// TIA Portal V19 export
FUNCTION "SUB_OUTPUT" : Void   // FC9, LAD
{ S7_Optimized_Access := 'TRUE' }
// stored: SetENOAutomatically false
BEGIN

REGION Network 1: "MGF FEED PUMP WORKING"
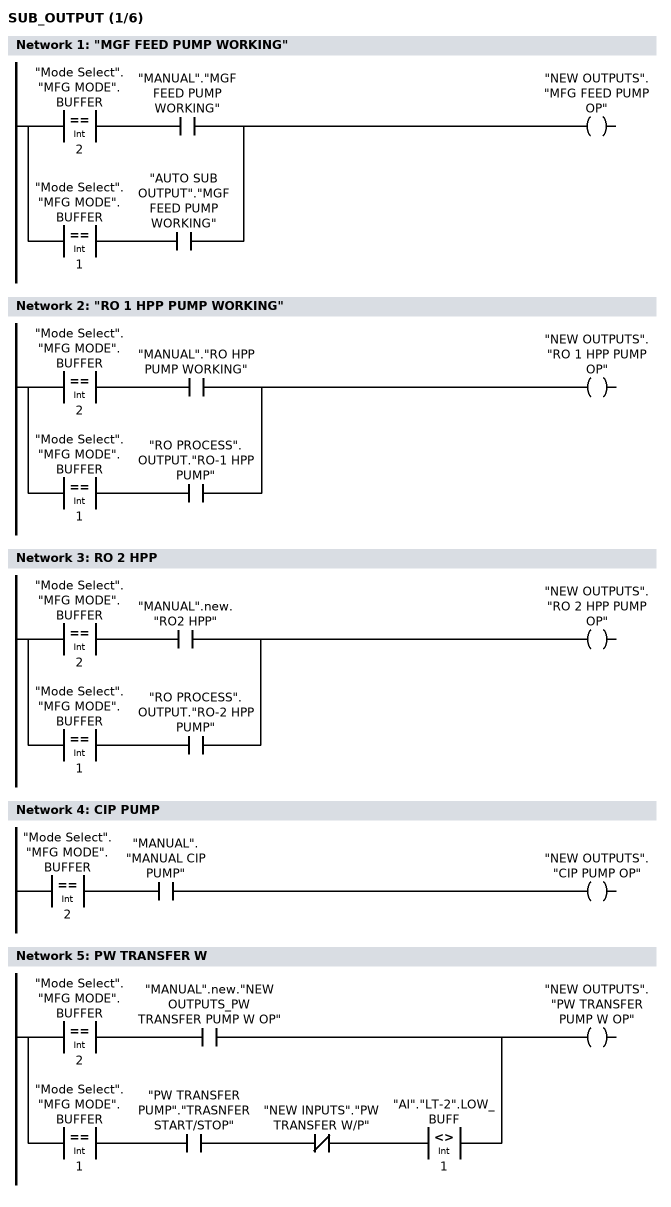
   RUNG wire#powerrail
      { S7_Templates := "SrcType := Int" } EQ_Contact(in1 := "Mode Select"."MFG MODE".BUFFER, in2 := 2)
      Contact( "MANUAL"."MGF FEED PUMP WORKING" )
      wire#w1
      Coil( "NEW OUTPUTS"."MFG FEED PUMP OP" )
   END_RUNG
   RUNG wire#powerrail
      { S7_Templates := "SrcType := Int" } EQ_Contact(in1 := "Mode Select"."MFG MODE".BUFFER, in2 := 1)
      Contact( "AUTO SUB OUTPUT"."MGF FEED PUMP WORKING" )
   END_RUNG wire#w1
   // the same network as SCL:
   "NEW OUTPUTS"."MFG FEED PUMP OP" := (("Mode Select"."MFG MODE".BUFFER = 2) AND "MANUAL"."MGF FEED PUMP WORKING") OR (("Mode Select"."MFG MODE".BUFFER = 1) AND "AUTO SUB OUTPUT"."MGF FEED PUMP WORKING");
END_REGION

REGION Network 2: "RO 1 HPP PUMP WORKING"
   RUNG wire#powerrail
      { S7_Templates := "SrcType := Int" } EQ_Contact(in1 := "Mode Select"."MFG MODE".BUFFER, in2 := 2)
      Contact( "MANUAL"."RO HPP PUMP WORKING" )
      wire#w1
      Coil( "NEW OUTPUTS"."RO 1 HPP PUMP OP" )
   END_RUNG
   RUNG wire#powerrail
      { S7_Templates := "SrcType := Int" } EQ_Contact(in1 := "Mode Select"."MFG MODE".BUFFER, in2 := 1)
      Contact( "RO PROCESS".OUTPUT."RO-1 HPP PUMP" )
   END_RUNG wire#w1
   // the same network as SCL:
   "NEW OUTPUTS"."RO 1 HPP PUMP OP" := (("Mode Select"."MFG MODE".BUFFER = 2) AND "MANUAL"."RO HPP PUMP WORKING") OR (("Mode Select"."MFG MODE".BUFFER = 1) AND "RO PROCESS".OUTPUT."RO-1 HPP PUMP");
END_REGION

REGION Network 3: RO 2 HPP
   RUNG wire#powerrail
      { S7_Templates := "SrcType := Int" } EQ_Contact(in1 := "Mode Select"."MFG MODE".BUFFER, in2 := 2)
      Contact( "MANUAL".new."RO2 HPP" )
      wire#w1
      Coil( "NEW OUTPUTS"."RO 2 HPP PUMP OP" )
   END_RUNG
   RUNG wire#powerrail
      { S7_Templates := "SrcType := Int" } EQ_Contact(in1 := "Mode Select"."MFG MODE".BUFFER, in2 := 1)
      Contact( "RO PROCESS".OUTPUT."RO-2 HPP PUMP" )
   END_RUNG wire#w1
   // the same network as SCL:
   "NEW OUTPUTS"."RO 2 HPP PUMP OP" := (("Mode Select"."MFG MODE".BUFFER = 2) AND "MANUAL".new."RO2 HPP") OR (("Mode Select"."MFG MODE".BUFFER = 1) AND "RO PROCESS".OUTPUT."RO-2 HPP PUMP");
END_REGION

REGION Network 4: CIP PUMP
   RUNG wire#powerrail
      { S7_Templates := "SrcType := Int" } EQ_Contact(in1 := "Mode Select"."MFG MODE".BUFFER, in2 := 2)
      Contact( "MANUAL"."MANUAL CIP PUMP" )
      Coil( "NEW OUTPUTS"."CIP PUMP OP" )
   END_RUNG
   // the same network as SCL:
   "NEW OUTPUTS"."CIP PUMP OP" := ("Mode Select"."MFG MODE".BUFFER = 2) AND "MANUAL"."MANUAL CIP PUMP";
END_REGION

REGION Network 5: PW TRANSFER W
   RUNG wire#powerrail
      { S7_Templates := "SrcType := Int" } EQ_Contact(in1 := "Mode Select"."MFG MODE".BUFFER, in2 := 2)
      Contact( "MANUAL".new."NEW OUTPUTS_PW TRANSFER PUMP W OP" )
      wire#w1
      Coil( "NEW OUTPUTS"."PW TRANSFER PUMP W OP" )
   END_RUNG
   RUNG wire#powerrail
      { S7_Templates := "SrcType := Int" } EQ_Contact(in1 := "Mode Select"."MFG MODE".BUFFER, in2 := 1)
      Contact( "PW TRANSFER PUMP"."TRASNFER START/STOP" )
      I_Contact( "NEW INPUTS"."PW TRANSFER W/P" )
      { S7_Templates := "SrcType := Int" } NE_Contact(in1 := "AI"."LT-2".LOW_BUFF, in2 := 1)
   END_RUNG wire#w1
   // the same network as SCL:
   "NEW OUTPUTS"."PW TRANSFER PUMP W OP" := (("Mode Select"."MFG MODE".BUFFER = 2) AND "MANUAL".new."NEW OUTPUTS_PW TRANSFER PUMP W OP") OR (("Mode Select"."MFG MODE".BUFFER = 1) AND "PW TRANSFER PUMP"."TRASNFER START/STOP" AND NOT "NEW INPUTS"."PW TRANSFER W/P" AND ("AI"."LT-2".LOW_BUFF <> 1));
END_REGION

REGION Network 6: PW TRANSFER S
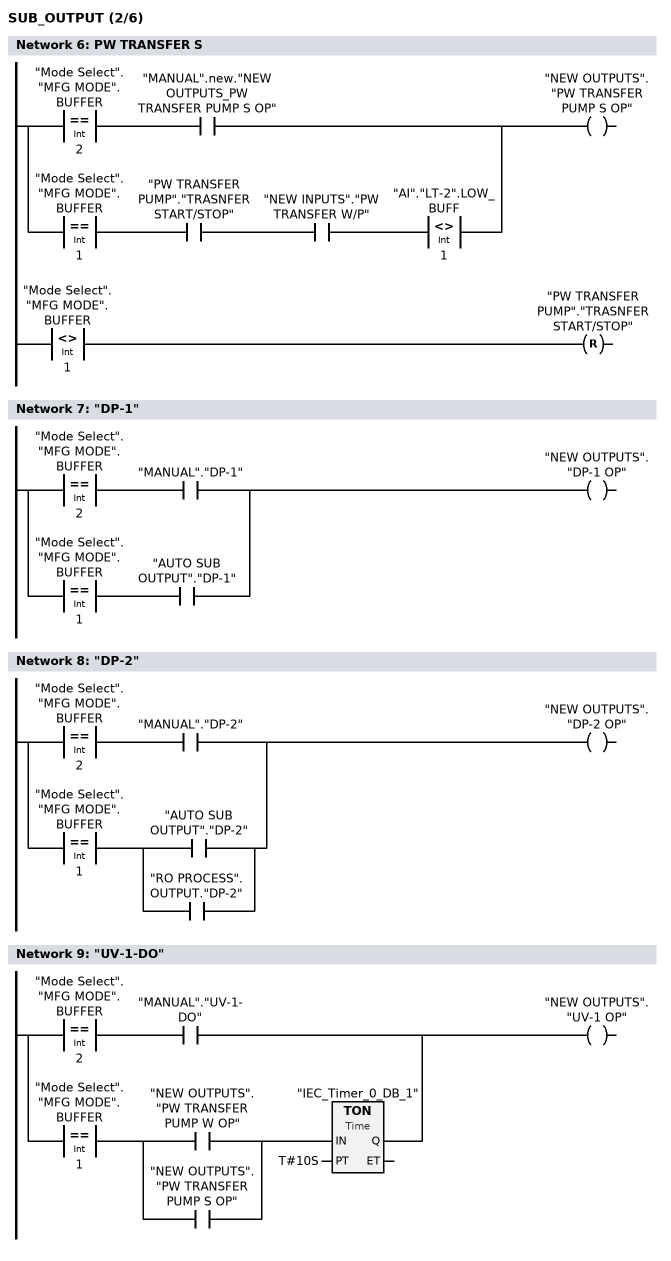
   RUNG wire#powerrail
      { S7_Templates := "SrcType := Int" } EQ_Contact(in1 := "Mode Select"."MFG MODE".BUFFER, in2 := 2)
      Contact( "MANUAL".new."NEW OUTPUTS_PW TRANSFER PUMP S OP" )
      wire#w1
      Coil( "NEW OUTPUTS"."PW TRANSFER PUMP S OP" )
   END_RUNG
   RUNG wire#powerrail
      { S7_Templates := "SrcType := Int" } EQ_Contact(in1 := "Mode Select"."MFG MODE".BUFFER, in2 := 1)
      Contact( "PW TRANSFER PUMP"."TRASNFER START/STOP" )
      Contact( "NEW INPUTS"."PW TRANSFER W/P" )
      { S7_Templates := "SrcType := Int" } NE_Contact(in1 := "AI"."LT-2".LOW_BUFF, in2 := 1)
   END_RUNG wire#w1
   RUNG wire#powerrail
      { S7_Templates := "SrcType := Int" } NE_Contact(in1 := "Mode Select"."MFG MODE".BUFFER, in2 := 1)
      R_Coil( "PW TRANSFER PUMP"."TRASNFER START/STOP" )
   END_RUNG
   // the same network as SCL:
   "NEW OUTPUTS"."PW TRANSFER PUMP S OP" := (("Mode Select"."MFG MODE".BUFFER = 2) AND "MANUAL".new."NEW OUTPUTS_PW TRANSFER PUMP S OP") OR (("Mode Select"."MFG MODE".BUFFER = 1) AND "PW TRANSFER PUMP"."TRASNFER START/STOP" AND "NEW INPUTS"."PW TRANSFER W/P" AND ("AI"."LT-2".LOW_BUFF <> 1));
   IF "Mode Select"."MFG MODE".BUFFER <> 1 THEN "PW TRANSFER PUMP"."TRASNFER START/STOP" := FALSE; END_IF;
END_REGION

REGION Network 7: "DP-1"
   RUNG wire#powerrail
      { S7_Templates := "SrcType := Int" } EQ_Contact(in1 := "Mode Select"."MFG MODE".BUFFER, in2 := 2)
      Contact( "MANUAL"."DP-1" )
      wire#w1
      Coil( "NEW OUTPUTS"."DP-1 OP" )
   END_RUNG
   RUNG wire#powerrail
      { S7_Templates := "SrcType := Int" } EQ_Contact(in1 := "Mode Select"."MFG MODE".BUFFER, in2 := 1)
      Contact( "AUTO SUB OUTPUT"."DP-1" )
   END_RUNG wire#w1
   // the same network as SCL:
   "NEW OUTPUTS"."DP-1 OP" := (("Mode Select"."MFG MODE".BUFFER = 2) AND "MANUAL"."DP-1") OR (("Mode Select"."MFG MODE".BUFFER = 1) AND "AUTO SUB OUTPUT"."DP-1");
END_REGION

REGION Network 8: "DP-2"
   RUNG wire#powerrail
      { S7_Templates := "SrcType := Int" } EQ_Contact(in1 := "Mode Select"."MFG MODE".BUFFER, in2 := 2)
      Contact( "MANUAL"."DP-2" )
      wire#w1
      Coil( "NEW OUTPUTS"."DP-2 OP" )
   END_RUNG
   RUNG wire#powerrail
      { S7_Templates := "SrcType := Int" } EQ_Contact(in1 := "Mode Select"."MFG MODE".BUFFER, in2 := 1)
      wire#w2
      Contact( "AUTO SUB OUTPUT"."DP-2" )
   END_RUNG wire#w1
   RUNG wire#w2
      Contact( "RO PROCESS".OUTPUT."DP-2" )
   END_RUNG wire#w1
   // the same network as SCL:
   "NEW OUTPUTS"."DP-2 OP" := (("Mode Select"."MFG MODE".BUFFER = 2) AND "MANUAL"."DP-2") OR (("Mode Select"."MFG MODE".BUFFER = 1) AND ("AUTO SUB OUTPUT"."DP-2" OR "RO PROCESS".OUTPUT."DP-2"));
END_REGION

REGION Network 9: "UV-1-DO"
   RUNG wire#powerrail
      { S7_Templates := "SrcType := Int" } EQ_Contact(in1 := "Mode Select"."MFG MODE".BUFFER, in2 := 2)
      Contact( "MANUAL"."UV-1-DO" )
      wire#w1
      Coil( "NEW OUTPUTS"."UV-1 OP" )
   END_RUNG
   RUNG wire#powerrail
      { S7_Templates := "SrcType := Int" } EQ_Contact(in1 := "Mode Select"."MFG MODE".BUFFER, in2 := 1)
      wire#w2
      Contact( "NEW OUTPUTS"."PW TRANSFER PUMP W OP" )
      wire#w3
      { S7_Templates := "time_type := Time" } "IEC_Timer_0_DB_1".TON(pt := T#10S, et =>)
   END_RUNG wire#w1
   RUNG wire#w2
      Contact( "NEW OUTPUTS"."PW TRANSFER PUMP S OP" )
   END_RUNG wire#w3
   // the same network as SCL:
   "IEC_Timer_0_DB_1".TON(IN := ("Mode Select"."MFG MODE".BUFFER = 1) AND ("NEW OUTPUTS"."PW TRANSFER PUMP W OP" OR "NEW OUTPUTS"."PW TRANSFER PUMP S OP"),
                          PT := T#10S);
   "NEW OUTPUTS"."UV-1 OP" := (("Mode Select"."MFG MODE".BUFFER = 2) AND "MANUAL"."UV-1-DO") OR "IEC_Timer_0_DB_1".Q;
END_REGION

REGION Network 10: "PSFV-1 – OPEN"
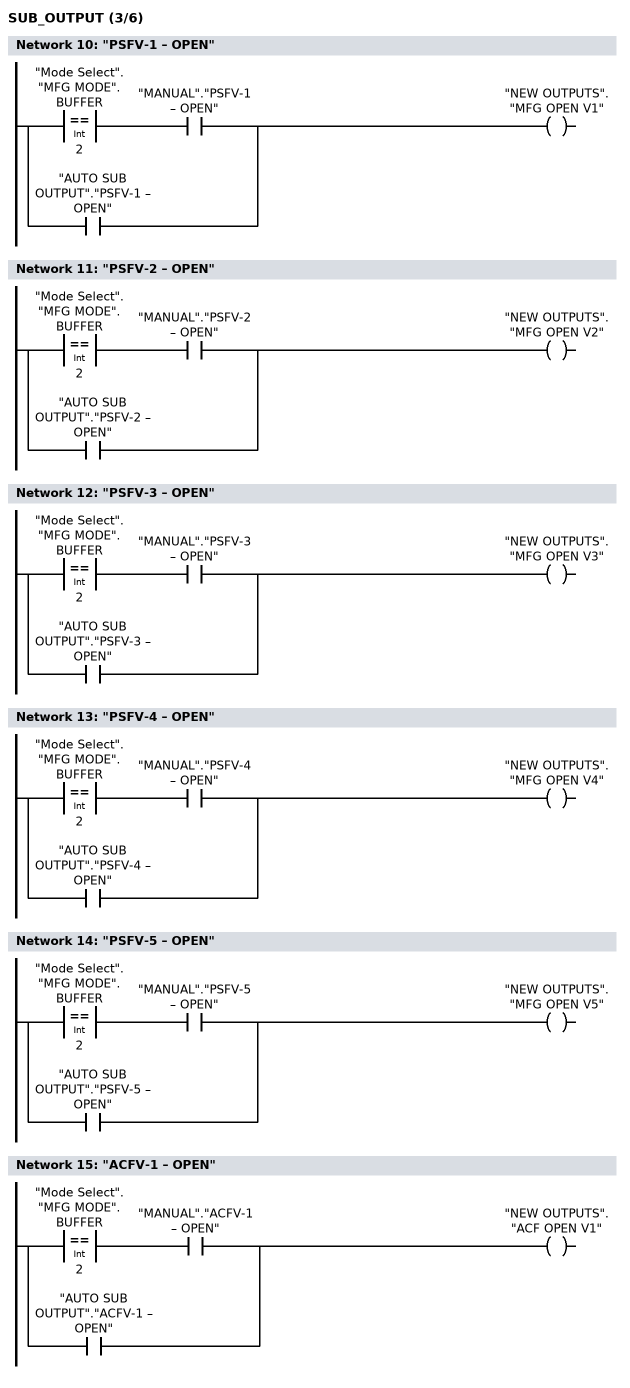
   RUNG wire#powerrail
      { S7_Templates := "SrcType := Int" } EQ_Contact(in1 := "Mode Select"."MFG MODE".BUFFER, in2 := 2)
      Contact( "MANUAL"."PSFV-1 – OPEN" )
      wire#w1
      Coil( "NEW OUTPUTS"."MFG OPEN V1" )
   END_RUNG
   RUNG wire#powerrail
      Contact( "AUTO SUB OUTPUT"."PSFV-1 – OPEN" )
   END_RUNG wire#w1
   // the same network as SCL:
   "NEW OUTPUTS"."MFG OPEN V1" := (("Mode Select"."MFG MODE".BUFFER = 2) AND "MANUAL"."PSFV-1 – OPEN") OR "AUTO SUB OUTPUT"."PSFV-1 – OPEN";
END_REGION

REGION Network 11: "PSFV-2 – OPEN"
   RUNG wire#powerrail
      { S7_Templates := "SrcType := Int" } EQ_Contact(in1 := "Mode Select"."MFG MODE".BUFFER, in2 := 2)
      Contact( "MANUAL"."PSFV-2 – OPEN" )
      wire#w1
      Coil( "NEW OUTPUTS"."MFG OPEN V2" )
   END_RUNG
   RUNG wire#powerrail
      Contact( "AUTO SUB OUTPUT"."PSFV-2 – OPEN" )
   END_RUNG wire#w1
   // the same network as SCL:
   "NEW OUTPUTS"."MFG OPEN V2" := (("Mode Select"."MFG MODE".BUFFER = 2) AND "MANUAL"."PSFV-2 – OPEN") OR "AUTO SUB OUTPUT"."PSFV-2 – OPEN";
END_REGION

REGION Network 12: "PSFV-3 – OPEN"
   RUNG wire#powerrail
      { S7_Templates := "SrcType := Int" } EQ_Contact(in1 := "Mode Select"."MFG MODE".BUFFER, in2 := 2)
      Contact( "MANUAL"."PSFV-3 – OPEN" )
      wire#w1
      Coil( "NEW OUTPUTS"."MFG OPEN V3" )
   END_RUNG
   RUNG wire#powerrail
      Contact( "AUTO SUB OUTPUT"."PSFV-3 – OPEN" )
   END_RUNG wire#w1
   // the same network as SCL:
   "NEW OUTPUTS"."MFG OPEN V3" := (("Mode Select"."MFG MODE".BUFFER = 2) AND "MANUAL"."PSFV-3 – OPEN") OR "AUTO SUB OUTPUT"."PSFV-3 – OPEN";
END_REGION

REGION Network 13: "PSFV-4 – OPEN"
   RUNG wire#powerrail
      { S7_Templates := "SrcType := Int" } EQ_Contact(in1 := "Mode Select"."MFG MODE".BUFFER, in2 := 2)
      Contact( "MANUAL"."PSFV-4 – OPEN" )
      wire#w1
      Coil( "NEW OUTPUTS"."MFG OPEN V4" )
   END_RUNG
   RUNG wire#powerrail
      Contact( "AUTO SUB OUTPUT"."PSFV-4 – OPEN" )
   END_RUNG wire#w1
   // the same network as SCL:
   "NEW OUTPUTS"."MFG OPEN V4" := (("Mode Select"."MFG MODE".BUFFER = 2) AND "MANUAL"."PSFV-4 – OPEN") OR "AUTO SUB OUTPUT"."PSFV-4 – OPEN";
END_REGION

REGION Network 14: "PSFV-5 – OPEN"
   RUNG wire#powerrail
      { S7_Templates := "SrcType := Int" } EQ_Contact(in1 := "Mode Select"."MFG MODE".BUFFER, in2 := 2)
      Contact( "MANUAL"."PSFV-5 – OPEN" )
      wire#w1
      Coil( "NEW OUTPUTS"."MFG OPEN V5" )
   END_RUNG
   RUNG wire#powerrail
      Contact( "AUTO SUB OUTPUT"."PSFV-5 – OPEN" )
   END_RUNG wire#w1
   // the same network as SCL:
   "NEW OUTPUTS"."MFG OPEN V5" := (("Mode Select"."MFG MODE".BUFFER = 2) AND "MANUAL"."PSFV-5 – OPEN") OR "AUTO SUB OUTPUT"."PSFV-5 – OPEN";
END_REGION

REGION Network 15: "ACFV-1 – OPEN"
   RUNG wire#powerrail
      { S7_Templates := "SrcType := Int" } EQ_Contact(in1 := "Mode Select"."MFG MODE".BUFFER, in2 := 2)
      Contact( "MANUAL"."ACFV-1 – OPEN" )
      wire#w1
      Coil( "NEW OUTPUTS"."ACF OPEN V1" )
   END_RUNG
   RUNG wire#powerrail
      Contact( "AUTO SUB OUTPUT"."ACFV-1 – OPEN" )
   END_RUNG wire#w1
   // the same network as SCL:
   "NEW OUTPUTS"."ACF OPEN V1" := (("Mode Select"."MFG MODE".BUFFER = 2) AND "MANUAL"."ACFV-1 – OPEN") OR "AUTO SUB OUTPUT"."ACFV-1 – OPEN";
END_REGION

REGION Network 16: "ACFV-2 – OPEN"
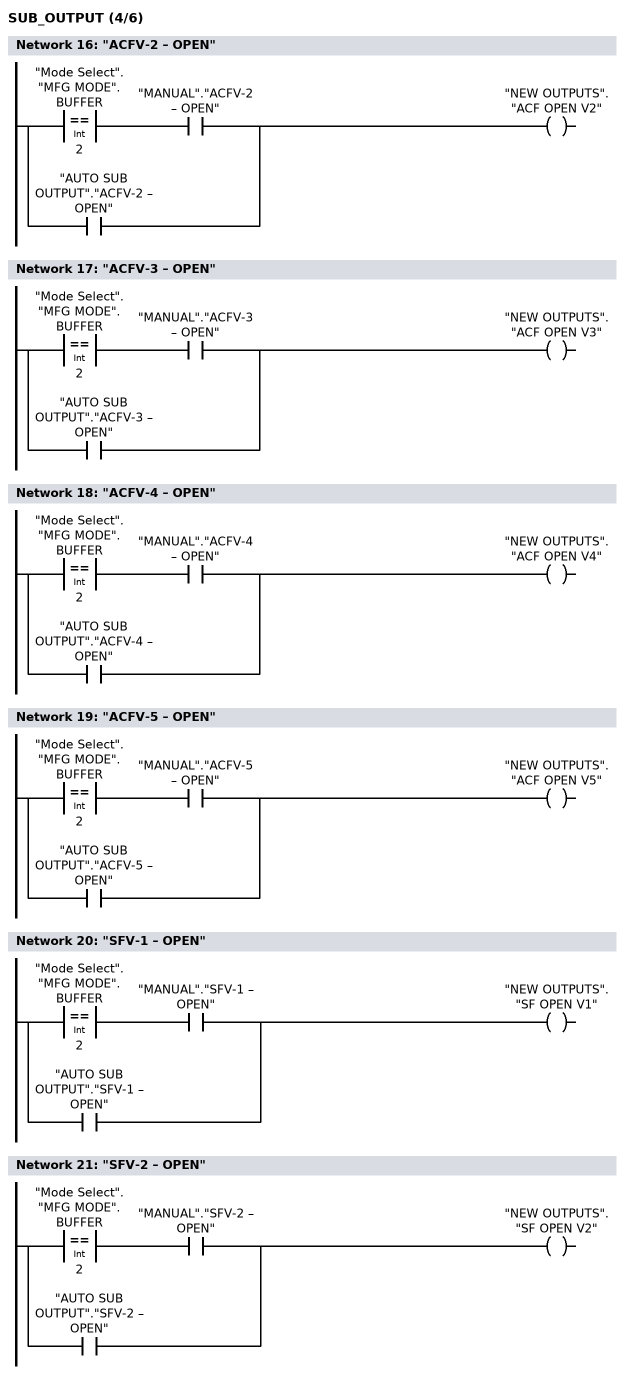
   RUNG wire#powerrail
      { S7_Templates := "SrcType := Int" } EQ_Contact(in1 := "Mode Select"."MFG MODE".BUFFER, in2 := 2)
      Contact( "MANUAL"."ACFV-2 – OPEN" )
      wire#w1
      Coil( "NEW OUTPUTS"."ACF OPEN V2" )
   END_RUNG
   RUNG wire#powerrail
      Contact( "AUTO SUB OUTPUT"."ACFV-2 – OPEN" )
   END_RUNG wire#w1
   // the same network as SCL:
   "NEW OUTPUTS"."ACF OPEN V2" := (("Mode Select"."MFG MODE".BUFFER = 2) AND "MANUAL"."ACFV-2 – OPEN") OR "AUTO SUB OUTPUT"."ACFV-2 – OPEN";
END_REGION

REGION Network 17: "ACFV-3 – OPEN"
   RUNG wire#powerrail
      { S7_Templates := "SrcType := Int" } EQ_Contact(in1 := "Mode Select"."MFG MODE".BUFFER, in2 := 2)
      Contact( "MANUAL"."ACFV-3 – OPEN" )
      wire#w1
      Coil( "NEW OUTPUTS"."ACF OPEN V3" )
   END_RUNG
   RUNG wire#powerrail
      Contact( "AUTO SUB OUTPUT"."ACFV-3 – OPEN" )
   END_RUNG wire#w1
   // the same network as SCL:
   "NEW OUTPUTS"."ACF OPEN V3" := (("Mode Select"."MFG MODE".BUFFER = 2) AND "MANUAL"."ACFV-3 – OPEN") OR "AUTO SUB OUTPUT"."ACFV-3 – OPEN";
END_REGION

REGION Network 18: "ACFV-4 – OPEN"
   RUNG wire#powerrail
      { S7_Templates := "SrcType := Int" } EQ_Contact(in1 := "Mode Select"."MFG MODE".BUFFER, in2 := 2)
      Contact( "MANUAL"."ACFV-4 – OPEN" )
      wire#w1
      Coil( "NEW OUTPUTS"."ACF OPEN V4" )
   END_RUNG
   RUNG wire#powerrail
      Contact( "AUTO SUB OUTPUT"."ACFV-4 – OPEN" )
   END_RUNG wire#w1
   // the same network as SCL:
   "NEW OUTPUTS"."ACF OPEN V4" := (("Mode Select"."MFG MODE".BUFFER = 2) AND "MANUAL"."ACFV-4 – OPEN") OR "AUTO SUB OUTPUT"."ACFV-4 – OPEN";
END_REGION

REGION Network 19: "ACFV-5 – OPEN"
   RUNG wire#powerrail
      { S7_Templates := "SrcType := Int" } EQ_Contact(in1 := "Mode Select"."MFG MODE".BUFFER, in2 := 2)
      Contact( "MANUAL"."ACFV-5 – OPEN" )
      wire#w1
      Coil( "NEW OUTPUTS"."ACF OPEN V5" )
   END_RUNG
   RUNG wire#powerrail
      Contact( "AUTO SUB OUTPUT"."ACFV-5 – OPEN" )
   END_RUNG wire#w1
   // the same network as SCL:
   "NEW OUTPUTS"."ACF OPEN V5" := (("Mode Select"."MFG MODE".BUFFER = 2) AND "MANUAL"."ACFV-5 – OPEN") OR "AUTO SUB OUTPUT"."ACFV-5 – OPEN";
END_REGION

REGION Network 20: "SFV-1 – OPEN"
   RUNG wire#powerrail
      { S7_Templates := "SrcType := Int" } EQ_Contact(in1 := "Mode Select"."MFG MODE".BUFFER, in2 := 2)
      Contact( "MANUAL"."SFV-1 – OPEN" )
      wire#w1
      Coil( "NEW OUTPUTS"."SF OPEN V1" )
   END_RUNG
   RUNG wire#powerrail
      Contact( "AUTO SUB OUTPUT"."SFV-1 – OPEN" )
   END_RUNG wire#w1
   // the same network as SCL:
   "NEW OUTPUTS"."SF OPEN V1" := (("Mode Select"."MFG MODE".BUFFER = 2) AND "MANUAL"."SFV-1 – OPEN") OR "AUTO SUB OUTPUT"."SFV-1 – OPEN";
END_REGION

REGION Network 21: "SFV-2 – OPEN"
   RUNG wire#powerrail
      { S7_Templates := "SrcType := Int" } EQ_Contact(in1 := "Mode Select"."MFG MODE".BUFFER, in2 := 2)
      Contact( "MANUAL"."SFV-2 – OPEN" )
      wire#w1
      Coil( "NEW OUTPUTS"."SF OPEN V2" )
   END_RUNG
   RUNG wire#powerrail
      Contact( "AUTO SUB OUTPUT"."SFV-2 – OPEN" )
   END_RUNG wire#w1
   // the same network as SCL:
   "NEW OUTPUTS"."SF OPEN V2" := (("Mode Select"."MFG MODE".BUFFER = 2) AND "MANUAL"."SFV-2 – OPEN") OR "AUTO SUB OUTPUT"."SFV-2 – OPEN";
END_REGION

REGION Network 22: "SFV-3 – OPEN"
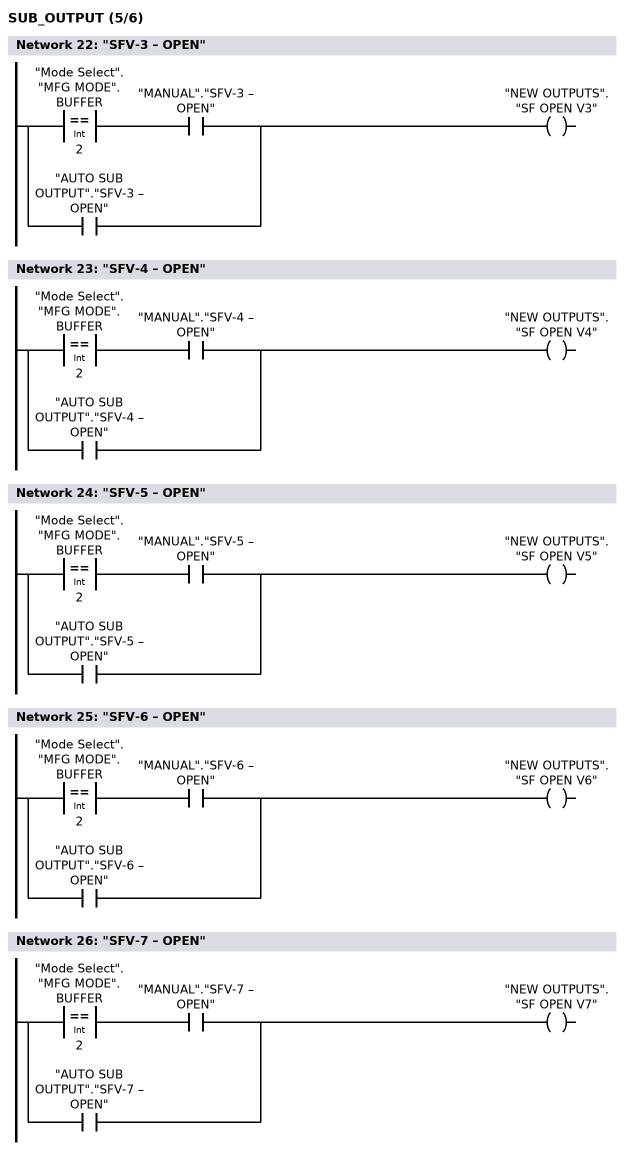
   RUNG wire#powerrail
      { S7_Templates := "SrcType := Int" } EQ_Contact(in1 := "Mode Select"."MFG MODE".BUFFER, in2 := 2)
      Contact( "MANUAL"."SFV-3 – OPEN" )
      wire#w1
      Coil( "NEW OUTPUTS"."SF OPEN V3" )
   END_RUNG
   RUNG wire#powerrail
      Contact( "AUTO SUB OUTPUT"."SFV-3 – OPEN" )
   END_RUNG wire#w1
   // the same network as SCL:
   "NEW OUTPUTS"."SF OPEN V3" := (("Mode Select"."MFG MODE".BUFFER = 2) AND "MANUAL"."SFV-3 – OPEN") OR "AUTO SUB OUTPUT"."SFV-3 – OPEN";
END_REGION

REGION Network 23: "SFV-4 – OPEN"
   RUNG wire#powerrail
      { S7_Templates := "SrcType := Int" } EQ_Contact(in1 := "Mode Select"."MFG MODE".BUFFER, in2 := 2)
      Contact( "MANUAL"."SFV-4 – OPEN" )
      wire#w1
      Coil( "NEW OUTPUTS"."SF OPEN V4" )
   END_RUNG
   RUNG wire#powerrail
      Contact( "AUTO SUB OUTPUT"."SFV-4 – OPEN" )
   END_RUNG wire#w1
   // the same network as SCL:
   "NEW OUTPUTS"."SF OPEN V4" := (("Mode Select"."MFG MODE".BUFFER = 2) AND "MANUAL"."SFV-4 – OPEN") OR "AUTO SUB OUTPUT"."SFV-4 – OPEN";
END_REGION

REGION Network 24: "SFV-5 – OPEN"
   RUNG wire#powerrail
      { S7_Templates := "SrcType := Int" } EQ_Contact(in1 := "Mode Select"."MFG MODE".BUFFER, in2 := 2)
      Contact( "MANUAL"."SFV-5 – OPEN" )
      wire#w1
      Coil( "NEW OUTPUTS"."SF OPEN V5" )
   END_RUNG
   RUNG wire#powerrail
      Contact( "AUTO SUB OUTPUT"."SFV-5 – OPEN" )
   END_RUNG wire#w1
   // the same network as SCL:
   "NEW OUTPUTS"."SF OPEN V5" := (("Mode Select"."MFG MODE".BUFFER = 2) AND "MANUAL"."SFV-5 – OPEN") OR "AUTO SUB OUTPUT"."SFV-5 – OPEN";
END_REGION

REGION Network 25: "SFV-6 – OPEN"
   RUNG wire#powerrail
      { S7_Templates := "SrcType := Int" } EQ_Contact(in1 := "Mode Select"."MFG MODE".BUFFER, in2 := 2)
      Contact( "MANUAL"."SFV-6 – OPEN" )
      wire#w1
      Coil( "NEW OUTPUTS"."SF OPEN V6" )
   END_RUNG
   RUNG wire#powerrail
      Contact( "AUTO SUB OUTPUT"."SFV-6 – OPEN" )
   END_RUNG wire#w1
   // the same network as SCL:
   "NEW OUTPUTS"."SF OPEN V6" := (("Mode Select"."MFG MODE".BUFFER = 2) AND "MANUAL"."SFV-6 – OPEN") OR "AUTO SUB OUTPUT"."SFV-6 – OPEN";
END_REGION

REGION Network 26: "SFV-7 – OPEN"
   RUNG wire#powerrail
      { S7_Templates := "SrcType := Int" } EQ_Contact(in1 := "Mode Select"."MFG MODE".BUFFER, in2 := 2)
      Contact( "MANUAL"."SFV-7 – OPEN" )
      wire#w1
      Coil( "NEW OUTPUTS"."SF OPEN V7" )
   END_RUNG
   RUNG wire#powerrail
      Contact( "AUTO SUB OUTPUT"."SFV-7 – OPEN" )
   END_RUNG wire#w1
   // the same network as SCL:
   "NEW OUTPUTS"."SF OPEN V7" := (("Mode Select"."MFG MODE".BUFFER = 2) AND "MANUAL"."SFV-7 – OPEN") OR "AUTO SUB OUTPUT"."SFV-7 – OPEN";
END_REGION

REGION Network 27: "AV-1 – OPEN"
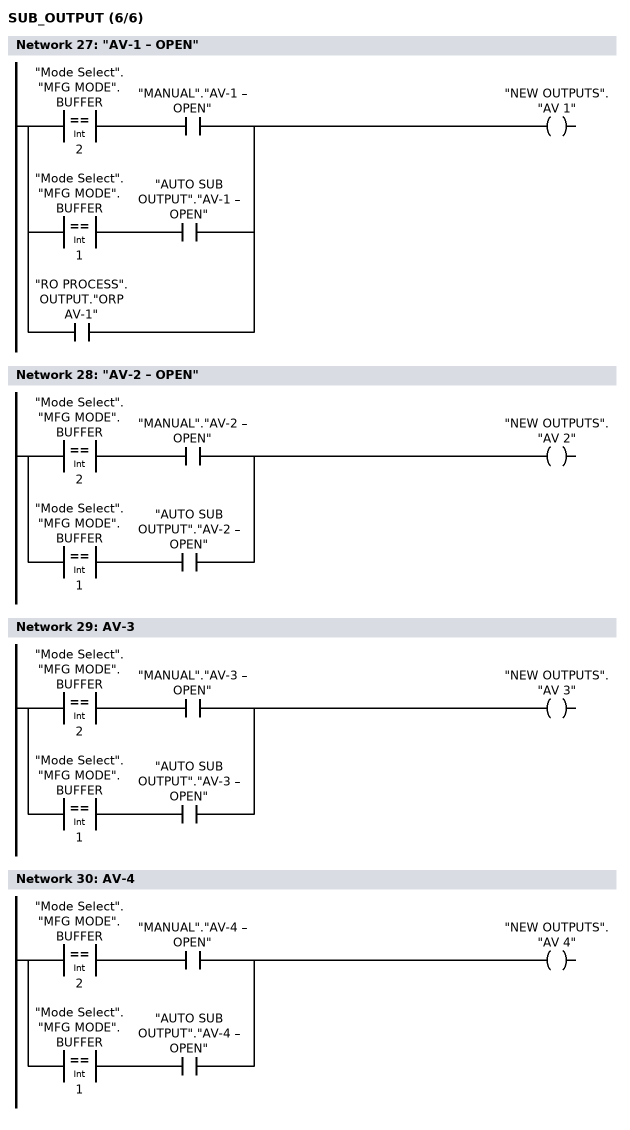
   RUNG wire#powerrail
      { S7_Templates := "SrcType := Int" } EQ_Contact(in1 := "Mode Select"."MFG MODE".BUFFER, in2 := 2)
      Contact( "MANUAL"."AV-1 – OPEN" )
      wire#w1
      Coil( "NEW OUTPUTS"."AV 1" )
   END_RUNG
   RUNG wire#powerrail
      { S7_Templates := "SrcType := Int" } EQ_Contact(in1 := "Mode Select"."MFG MODE".BUFFER, in2 := 1)
      Contact( "AUTO SUB OUTPUT"."AV-1 – OPEN" )
   END_RUNG wire#w1
   RUNG wire#powerrail
      Contact( "RO PROCESS".OUTPUT."ORP AV-1" )
   END_RUNG wire#w1
   // the same network as SCL:
   "NEW OUTPUTS"."AV 1" := (("Mode Select"."MFG MODE".BUFFER = 2) AND "MANUAL"."AV-1 – OPEN") OR (("Mode Select"."MFG MODE".BUFFER = 1) AND "AUTO SUB OUTPUT"."AV-1 – OPEN") OR "RO PROCESS".OUTPUT."ORP AV-1";
END_REGION

REGION Network 28: "AV-2 – OPEN"
   RUNG wire#powerrail
      { S7_Templates := "SrcType := Int" } EQ_Contact(in1 := "Mode Select"."MFG MODE".BUFFER, in2 := 2)
      Contact( "MANUAL"."AV-2 – OPEN" )
      wire#w1
      Coil( "NEW OUTPUTS"."AV 2" )
   END_RUNG
   RUNG wire#powerrail
      { S7_Templates := "SrcType := Int" } EQ_Contact(in1 := "Mode Select"."MFG MODE".BUFFER, in2 := 1)
      Contact( "AUTO SUB OUTPUT"."AV-2 – OPEN" )
   END_RUNG wire#w1
   // the same network as SCL:
   "NEW OUTPUTS"."AV 2" := (("Mode Select"."MFG MODE".BUFFER = 2) AND "MANUAL"."AV-2 – OPEN") OR (("Mode Select"."MFG MODE".BUFFER = 1) AND "AUTO SUB OUTPUT"."AV-2 – OPEN");
END_REGION

REGION Network 29: AV-3
   RUNG wire#powerrail
      { S7_Templates := "SrcType := Int" } EQ_Contact(in1 := "Mode Select"."MFG MODE".BUFFER, in2 := 2)
      Contact( "MANUAL"."AV-3 – OPEN" )
      wire#w1
      Coil( "NEW OUTPUTS"."AV 3" )
   END_RUNG
   RUNG wire#powerrail
      { S7_Templates := "SrcType := Int" } EQ_Contact(in1 := "Mode Select"."MFG MODE".BUFFER, in2 := 1)
      Contact( "AUTO SUB OUTPUT"."AV-3 – OPEN" )
   END_RUNG wire#w1
   // the same network as SCL:
   "NEW OUTPUTS"."AV 3" := (("Mode Select"."MFG MODE".BUFFER = 2) AND "MANUAL"."AV-3 – OPEN") OR (("Mode Select"."MFG MODE".BUFFER = 1) AND "AUTO SUB OUTPUT"."AV-3 – OPEN");
END_REGION

REGION Network 30: AV-4
   RUNG wire#powerrail
      { S7_Templates := "SrcType := Int" } EQ_Contact(in1 := "Mode Select"."MFG MODE".BUFFER, in2 := 2)
      Contact( "MANUAL"."AV-4 – OPEN" )
      wire#w1
      Coil( "NEW OUTPUTS"."AV 4" )
   END_RUNG
   RUNG wire#powerrail
      { S7_Templates := "SrcType := Int" } EQ_Contact(in1 := "Mode Select"."MFG MODE".BUFFER, in2 := 1)
      Contact( "AUTO SUB OUTPUT"."AV-4 – OPEN" )
   END_RUNG wire#w1
   // the same network as SCL:
   "NEW OUTPUTS"."AV 4" := (("Mode Select"."MFG MODE".BUFFER = 2) AND "MANUAL"."AV-4 – OPEN") OR (("Mode Select"."MFG MODE".BUFFER = 1) AND "AUTO SUB OUTPUT"."AV-4 – OPEN");
END_REGION
END_FUNCTION
